PROGRAM OP110_Initialization_Seq
VAR
END_VAR

IF (SR110_Vert_servo_ctrl.Axis_In_Home)THEN
OP20_Temp_hmeOK:=TRUE;
OP20_HomeRunning:=FALSE;
OP20_Homing_Seq:=0;
ELSE
	OP20_Temp_hmeOK:=FALSE;	
END_IF

CASE OP20_Homing_Seq OF
	0: IF (OP20_AutoSelected AND NOT OP20_HomeRunning AND NOT OP20_ErrorActive AND NOT OP20_AutoRunning AND NOT OP20_StepRunning AND NOT OP20_Temp_hmeOK) THEN
		OP20_HomeRunning:=TRUE;
		OP20_Homing_Seq:=10;	
	   END_IF
	10:IF (OP20_HomeRunning AND OP20_HMI_Homing)THEN 
		IF (SR110_Vert_servo_ctrl.Axis_In_Home) THEN 
			//OP20_Homing_Seq:=20;
			SR110_Vert_servo_ctrl.Axis_Home_Cmd:=FALSE;
		ELSE
			SR110_Vert_servo_ctrl.Axis_Home_Cmd:=TRUE;
	    END_IF
		OP20_Homing_Seq:=20;
	   END_IF		
	20:	OP20_Homing_Seq:=0;
		OP20_HomeRunning:=FALSE;
		OP20_HMI_Homing:=FALSE;
END_CASE

END_PROGRAM

(* stored: Version 1.1.0.1, ProductVersion 3.1.4024.11
   POU OP110_Initialization_Seq: Id {44aa57e4-bd66-401d-91ab-328dbea3e0de}, SpecialFunc None *)
